// Mitsubishi GX Works2 project: 인터록 자기유지 통합 회로   PLC: Q03UDV

PROGRAM MAIN
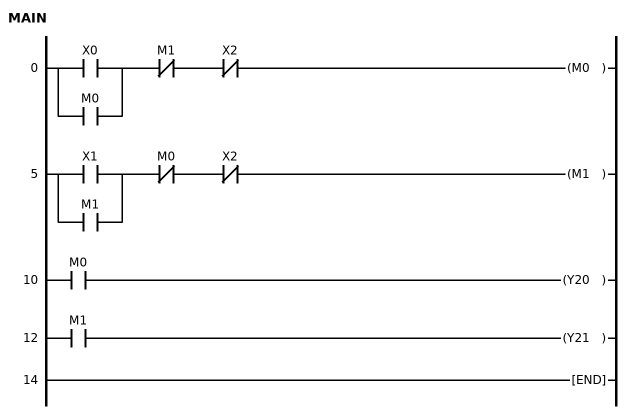
0     LD      X0
      OR      M0
      ANI     M1
      ANI     X2
      OUT     M0
5     LD      X1
      OR      M1
      ANI     M0
      ANI     X2
      OUT     M1
10    LD      M0
      OUT     Y20
12    LD      M1
      OUT     Y21
14    END
END_PROGRAM
